PROGRAM MAIN
VAR		

END_VAR

IF GV_LIFT.DOOR_1_INDICATOR_LATCH_IN THEN
	GV_LIFT.DOOR_1_INDICATOR_LATCH_OUT := TRUE;
ELSE
	GV_LIFT.DOOR_1_INDICATOR_LATCH_OUT := FALSE;	
END_IF

IF GV_LIFT.PIT_ESTOP_INDICATOR_IN THEN
	GV_LIFT.PIT_ESTOP_INDICATOR_OUT := TRUE;
ELSE
	GV_LIFT.PIT_ESTOP_INDICATOR_OUT := FALSE;	
END_IF

IF GV_LIFT.DOWNSTAGE_ESTOP_INDICATOR_IN THEN
	GV_LIFT.DOWNSTAGE_ESTOP_INDICATOR_OUT := TRUE;
ELSE
	GV_LIFT.DOWNSTAGE_ESTOP_INDICATOR_OUT := FALSE;	
END_IF

IF GV_LIFT.ESTOP_INDICATOR_IN THEN
	GV_LIFT.ESTOP_INDICATOR_OUT := TRUE;
ELSE
	GV_LIFT.ESTOP_INDICATOR_OUT := FALSE;	
END_IF

IF GV_LIFT.FAULT_INDICATOR_IN THEN
	GV_LIFT.FAULT_INDICATOR_OUT := TRUE;
ELSE
	GV_LIFT.FAULT_INDICATOR_OUT := FALSE;	
END_IF

IF GV_LIFT.UP_BUTTON_IN THEN
	GV_LIFT.UP_BUTTON_OUT := TRUE;
ELSE
	GV_LIFT.UP_BUTTON_OUT := FALSE;
END_IF

IF GV_LIFT.DOWN_BUTTON_IN THEN
	GV_LIFT.DOWN_BUTTON_OUT := TRUE;
ELSE
	GV_LIFT.DOWN_BUTTON_OUT := FALSE;
END_IF

IF GV_LIFT.RUN_BUTTON_IN THEN
	GV_LIFT.RUN_BUTTON_OUT := TRUE;
ELSE
	GV_LIFT.RUN_BUTTON_OUT := FALSE;
END_IF

XML(); 
HMI();
IO_SWITCHBOARD();
SYSTEM_RESET();
MOVE_TO_POSITION();
SwitchScreens();

END_PROGRAM

(* stored: Version 1.1.0.1, ProductVersion 3.1.4022.12
   POU MAIN: Id {f931fcee-5ac4-4068-9063-b3a0ff76f962}, SpecialFunc None *)
